// TIA Portal V17 export
// export: Created 2021-12-03T08:13:01.1583031Z, ExportSetting WithDefaults, DisplayName Totally Integrated Automation Portal, DisplayVersion V17, DisplayName TIA Portal Openness, DisplayVersion V17, DisplayName TIA Portal Version Control Interface, DisplayVersion V17, DisplayName STEP 7 Professional, DisplayVersion V17, DisplayName STEP 7 Safety, DisplayVersion V17, DisplayName WinCC Advanced, DisplayVersion V17
DATA_BLOCK "GDB_ScanSequence"   // DB17
VERSION : 0.1
// stored: AutoNumber true, IsOnlyStoredInLoadMemory false, IsWriteProtectedInAS false
   VAR
      Run : Bool;   // Цикл
      IntrptCycl : Bool;   // Цикл прерван
      RdyForScan : Bool;   // Готовность комплекса к сканированию
      DetLineRdy : Bool;   // Готовность детекторной линейки
      AccRdy : Bool;   // Готовность ускорителя
      ConvRdy : Bool;   // Конвейер готов
      ScanSpNr : Int;
      SR : Struct
         Run : Bool;
         BwdDetLineStp : Bool;
         FwdDetLineStp : Bool;
      END_STRUCT;
      N_TRIG : Struct
         BwdDetLineStp : Bool;
         FwdDetLineStp : Bool;
      END_STRUCT;
      Transit : Struct   // Переходы
         Strt : Bool;   // Старт
         StrtHomming : Bool;   // Старт с возвратом в домашнюю позицию
         HomPosit : Bool;   // Конвейер в домашней позиции
         PrepareDelay : Bool;   // Задержка в шаге подготовка
         WithOutAcc : Bool;   // Без ускорителя
         WithRfOn : Bool;   // С СВЧ
         WithOutRfOn : Bool;   // Без СВЧ
         DelayRF : Bool;   // Задержка после включения RF
         DelayXray : Bool;   // Задержка после включения XRay
         FwdPos : Bool;   // В конечной позиции FWD
         BwdPos : Bool;   // В конечной позиции BWD
         BwdDetLineStrt : Bool;   // Старт детекторной линейки при движении BWD
         BwdDetLineStp : Bool;   // Стоп детекторной линейки при движении BWD
         FwdDetLineStrt : Bool;   // Старт детекторной линейки при движении FWD
         FwdDetLineStp : Bool;   // Стоп детекторной линейки при движении FWD
         EndPosition : Bool;   // Конечная позиция
         ScanCompl : Bool;   // Сканирование завершено
      END_STRUCT;
      Action : Struct   // Действия
         Prepare : Bool;   // Подготовка
         BwdMoveReq : Bool;   // Старт для движения назад
         FwdMoveReq : Bool;   // Старт для движения вперед
         DetLineStrtReq : Bool;   // Старт детекторной линейки
         DetLineStpReq : Bool;   // Стоп детекторной линейки
         RfOnReq : Bool;   // Запрос на включение RfOn
         XrayOnReq : Bool;   // Запрос на включение XrayOn
         ScanCompl : Bool;
      END_STRUCT;
      "Step" : Struct   // Шаги
         Preparation : Bool;   // Подготовка
         RF_On : Bool;   // СВЧ
         XRay_On : Bool;   // Тормозное излучение
         Homing : Bool;
         StrtMove : Bool;   // Начало движения
         Scanning : Bool;   // Сканирование
         EndMove : Bool;   // Окончание движения
         ScanCompl : Bool;   // Сканирование завершено
      END_STRUCT;
   END_VAR
BEGIN
END_DATA_BLOCK
